FUNCTION_BLOCK ClearLinkEIP_old
VAR_INPUT
	bEnable : BOOL;
END_VAR
VAR_OUTPUT
	pulse AT %Q* : INT; //num pulses
	outputRegister AT %Q* : INT;
	brakeRelease AT %Q* : BOOL;
	
	A : BOOL; //direction (F = inwards, T = outwards)
	B : BOOL; //home bit
	clear : BOOL; //clear error
	
	contact AT %I* : BOOL;
	home AT %I* : BOOL;
	outerLimit AT %I* : BOOL;
	innerLimit AT %I* : BOOL;
	
	hlfb AT %I* : REAL;
	
	homeSet : BOOL;
	busy : BOOL;
	error : BOOL;
	
	position : LREAL;
	targetPos : LREAL;
END_VAR
VAR
	pulseRequest : INT;
	pulser : TON;
	
	minHoming : TON;
	resetTimer : TP;
	errorTimer : TON;
	
	step : Homing; //(IDLE, HOME_UP, HOME_FINAL, DOWN, REDO_HOME, HOME_DONE);
	mode : (DISABLE, HOLD, TARGET, CONTINUOUS, RESET_ERR);
END_VAR
VAR_STAT CONSTANT
	resetTime : TIME := T#1000MS;
	errorTime : TIME := T#1000MS;
	unitsPerPulse : INT := 800; //800 Teknic units per revolution
	distancePerPulse : INT := 5; //5mm per revolution
END_VAR

(*
public motion methods should not directly access the motion variables
they should only modify the mode, which this FB will then validate based on its internal parameters
*)


IF NOT bEnable THEN
	mode := DISABLE;
END_IF

outputRegister.0 := bEnable;
outputRegister.1 := A;
outputRegister.2 := B;
outputRegister.3 := clear;

resetTimer(IN:= , PT:= resetTime, Q=> clear, ET=> );
errorTimer(IN:= , PT:= errorTime, Q=> error, ET=> );

//set the bool outputs, all are listed for readability
homeSet := homeSet;
busy := hlfb <> -9999;
error := error;

IF home AND_THEN A THEN //block outwards motion
	position := 0;
	pulse := 0;
	pulseRequest := 0;
	mode := HOLD;
(*
ELSIF outerLimit AND_THEN A THEN //block outwards motion
	mode := HOLD;

ELSIF innerLimit AND_THEN NOT A THEN //block inwards motion
	mode := HOLD;
*)
ELSIF
	(outerLimit AND A) OR //block outwards motion
	(innerLimit AND NOT A) //block inwards motion
THEN
	mode := HOLD;
END_IF


CASE mode OF
	DISABLE:
		//bEnable := FALSE;
		pulse := 0;
		pulseRequest := 0;
		
	HOLD:
		pulse := 0;
		pulseRequest := 0;
	
	TARGET:
		IF WithinTolerance(position, targetPos, distancePerPulse) THEN
			pulseRequest := 0;
			mode := HOLD;
			
		ELSIF NOT busy THEN //pulseRequest is only taken if motor is not running, so requests > 1 should not stack
			A :=  position < targetPos;
			pulseRequest := TO_INT(ABS(position - targetPos)/distancePerPulse);
			//pulseRequest := 1;
			
		END_IF
		
	CONTINUOUS:
		pulseRequest := 1;
		
	RESET_ERR:
		pulse := 0;
		pulseRequest := 0;
		resetTimer.IN := TRUE;
		
		IF resetTimer.Q THEN
			resetTimer.IN := FALSE;
			mode := HOLD;
		END_IF
		
END_CASE

sequence();

METHOD homingSequence : BOOL
minHoming(IN:= , PT:= T#1S, Q=> , ET=> );

IF NOT bEnable THEN
	mode := DISABLE;
	RETURN;
END_IF

CASE step OF
	Homing.IDLE:
		A := FALSE;
		B := FALSE;
		brakeRelease := TRUE;
		
		homeSet := FALSE;
		step := Homing.REDO;
		
	Homing.REDO: //let insertion drop to inner limit before homing
		A := FALSE;
		B := FALSE;
		brakeRelease := TRUE;
		
		IF NOT innerLimit THEN
			mode := CONTINUOUS;
			step := Homing.HOME_OUT;
		END_IF
	
	Homing.HOME_OUT:
		mode := CONTINUOUS;
	
		A := FALSE;
		B := TRUE;
		brakeRelease := TRUE;
		
		minHoming.IN := TRUE;
		
		IF NOT home AND minHoming.Q THEN
			minHoming.IN := FALSE;
			
			mode := HOLD;
			step := Homing.DONE;
		END_IF
		
	Homing.DONE:
		pulse := 0;
		A := FALSE;
		B := FALSE;
		brakeRelease := TRUE;
		
		position := 0;
		homeSet := TRUE;
		homingSequence := TRUE;
		
		mode := HOLD;
		step := Homing.IDLE;
	
END_CASE
END_METHOD

METHOD moveAbsolute : BOOL
VAR_INPUT
	newTarget : LREAL;
END_VAR
targetPos := newTarget;
mode := TARGET;
END_METHOD

METHOD moveContinuous : BOOL
VAR_INPUT
	direction : MC_Direction;
END_VAR
IF direction = MC_Negative_Direction THEN
	A := FALSE;
ELSIF direction = MC_Positive_Direction THEN
	A := TRUE;
END_IF

mode := CONTINUOUS;
END_METHOD

METHOD reset : BOOL
VAR_INPUT
END_VAR
mode := RESET_ERR;
errorTimer.IN := FALSE;
END_METHOD

METHOD sequence : BOOL
VAR_INPUT
END_VAR
IF pulse > 0 AND hlfb = -9999 THEN //no response, start error timer
	errorTimer.IN := TRUE;
	
ELSIF hlfb > -9999 THEN //pulses received
	errorTimer.IN := FALSE;
	IF A THEN //positive
		position := position + (distancePerPulse * pulse);
	ELSE
		position := position - (distancePerPulse * pulse);
	END_IF
	pulse := 0;
	RETURN;
END_IF

//is free to accept new request
IF pulse = 0 (*AND NOT pulseSeparator.Q*) THEN
	pulse := pulseRequest;
	//pulseRequest := 0;
END_IF
END_METHOD

METHOD stop : BOOL
VAR_INPUT
END_VAR
mode := HOLD;
END_METHOD

END_FUNCTION_BLOCK

(* stored: Version 1.1.0.1, ProductVersion 3.1.4024.11
   POU ClearLinkEIP_old: Id {1d47033b-d774-42fe-b022-c8ddd8488a6f}, SpecialFunc None
   Folder Public Methods: Id {d29c5c5d-14f1-4972-8db5-81b3764b5246}
   Method homingSequence: Id {925d6ae9-57fa-4c20-b488-bf8b58e8f70a}
   Method moveAbsolute: Id {48d9973d-9fcb-433c-b03e-e671dd2fbe37}
   Method moveContinuous: Id {32b5f905-3046-435e-bedb-532126f570d4}
   Method reset: Id {a54fb6bd-1435-4800-ad76-8a72a5bacf80}
   Method sequence: Id {4fdb4002-c74d-4629-b33e-bcb75c287ea7}
   Method stop: Id {93d5c5d8-8608-4ab9-806f-64dab48570ea} *)
